PROGRAM MAIN
VAR
	nIndex AT %I*		:	DINT;
	sText AT %I*		:	T_MaxString;
	nLen				:	DINT;
END_VAR

nlen := len(sText);

END_PROGRAM

(* stored: Version 1.1.0.1, ProductVersion 3.1.4024.5
   POU MAIN: Id {cce82f76-8d03-4165-a818-ad2af920b87d}, SpecialFunc None *)
